VAR_GLOBAL CONSTANT
	CARRIAGE_RETURN : BYTE := 16#D;
	LINE_FEED : BYTE := 16#A;
	ASCI_SEMI_COLON : BYTE := 16#3B;
	ASCI_COMMA		: BYTE := 16#2C;
END_VAR

(* stored: Version 1.1.0.1, ProductVersion 3.1.4022.12
   GVL Character: Id {6524787a-9b6c-4eb5-95be-b8cb40a5bf0f} *)
